# EPICS autosave request: ADPSL/pslApp/Db/PSL_settings.req
$(P)$(R)CameraName
$(P)$(R)TIFFComment
